// TIA Portal V18 export
// export: Created 2026-06-08T16:32:21.5795508Z, ExportSetting WithDefaults, DisplayName Totally Integrated Automation Portal, DisplayVersion V18, DisplayName TIA Portal Openness, DisplayVersion V18, DisplayName TIA Portal Version Control Interface, DisplayVersion V18, DisplayName STEP 7 Professional, DisplayVersion V18, DisplayName STEP 7 Safety, DisplayVersion V18, DisplayName WinCC Professional, DisplayVersion V18
FUNCTION_BLOCK "Assembly_Emergency"   // FB13, LAD
VERSION : 0.1
// stored: AutoNumber true, IsIECCheckEnabled false, UDAEnableTagReadback false
BEGIN

REGION Network 1
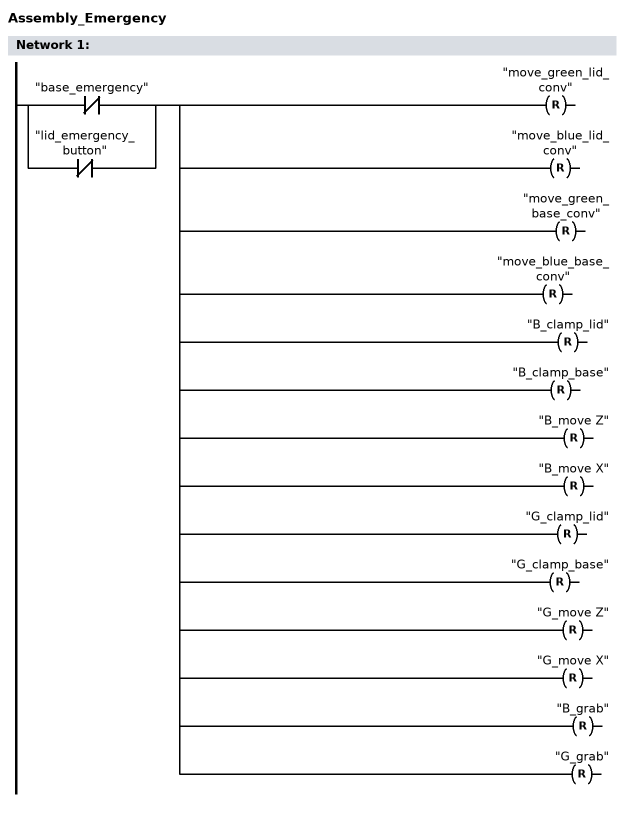
   RUNG wire#powerrail
      I_Contact( "base_emergency" )
      wire#w1
      R_Coil( "move_green_lid_conv" )
   END_RUNG
   RUNG wire#powerrail
      I_Contact( "lid_emergency_button" )
   END_RUNG wire#w1
   RUNG wire#w1
      R_Coil( "move_blue_lid_conv" )
   END_RUNG
   RUNG wire#w1
      R_Coil( "move_green_base_conv" )
   END_RUNG
   RUNG wire#w1
      R_Coil( "move_blue_base_conv" )
   END_RUNG
   RUNG wire#w1
      R_Coil( "B_clamp_lid" )
   END_RUNG
   RUNG wire#w1
      R_Coil( "B_clamp_base" )
   END_RUNG
   RUNG wire#w1
      R_Coil( "B_move Z" )
   END_RUNG
   RUNG wire#w1
      R_Coil( "B_move X" )
   END_RUNG
   RUNG wire#w1
      R_Coil( "G_clamp_lid" )
   END_RUNG
   RUNG wire#w1
      R_Coil( "G_clamp_base" )
   END_RUNG
   RUNG wire#w1
      R_Coil( "G_move Z" )
   END_RUNG
   RUNG wire#w1
      R_Coil( "G_move X" )
   END_RUNG
   RUNG wire#w1
      R_Coil( "B_grab" )
   END_RUNG
   RUNG wire#w1
      R_Coil( "G_grab" )
   END_RUNG
   // the same network as SCL:
   IF NOT "base_emergency" OR NOT "lid_emergency_button" THEN
       "move_green_lid_conv" := FALSE;
       "move_blue_lid_conv" := FALSE;
       "move_green_base_conv" := FALSE;
       "move_blue_base_conv" := FALSE;
       "B_clamp_lid" := FALSE;
       "B_clamp_base" := FALSE;
       "B_move Z" := FALSE;
       "B_move X" := FALSE;
       "G_clamp_lid" := FALSE;
       "G_clamp_base" := FALSE;
       "G_move Z" := FALSE;
       "G_move X" := FALSE;
       "B_grab" := FALSE;
       "G_grab" := FALSE;
   END_IF;
END_REGION
END_FUNCTION_BLOCK
